FUNCTION_BLOCK DualHysteresis_AR_AX (* 2-way conversion of Analog to Digital with Hysteresis (Switch-on = MI +/- (ABS(DEAD) + ABS(HYSTERESIS)), Switch-off = MI +/- ABS(DEAD)) *)
  (* Standard: 61499-2; Description: Copyright (c) 2023 HR Agrartechnik GmbH This program and the accompanying materials are made available under the terms of the Eclipse Public License 2.0 which is available at https://www.eclipse.org/legal/epl-2.0/ SPDX-License-Identifier: EPL-2.0 *)
  (* Version 3.1, 2026-06-01, Gemini CLI, Addressed code review: absolute values for thresholds, explicit comparison semantics. *)
  (* Version 3.0, 2025-04-14, Patrick Aigner, changed package *)
  (* Version 1.0, 2023-06-06, Franz Höpfinger, HR Agrartechnik GmbH *)
  PACKAGE logiBUS::signalprocessing::hysteresis;
  IMPORT eclipse4diac::core::TypeHash;
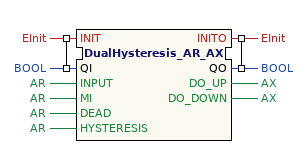
  EVENT_INPUT
    INIT : EInit WITH QI; (* Initialization Request *)
  END_EVENT
  EVENT_OUTPUT
    INITO : EInit WITH QO; (* Initialization Confirm *)
  END_EVENT
  VAR_INPUT
    QI : BOOL; (* Input event qualifier *)
  END_VAR
  VAR_OUTPUT
    QO : BOOL;
  END_VAR
  SOCKETS
    INPUT : adapter::types::unidirectional::AR; (* Input value *)
    MI : adapter::types::unidirectional::AR; (* Center point (e.g. 0.5 for 50%) *)
    DEAD : adapter::types::unidirectional::AR; (* Deadband around MI (absolute value). Switch-off points = MI +/- ABS(DEAD) *)
    HYSTERESIS : adapter::types::unidirectional::AR; (* Hysteresis value (absolute value). Switch-on points = MI +/- (ABS(DEAD) + ABS(HYSTERESIS)) *)
  END_SOCKETS
  PLUGS
    DO_UP : adapter::types::unidirectional::AX; (* UP *)
    DO_DOWN : adapter::types::unidirectional::AX; (* DOWN *)
  END_PLUGS
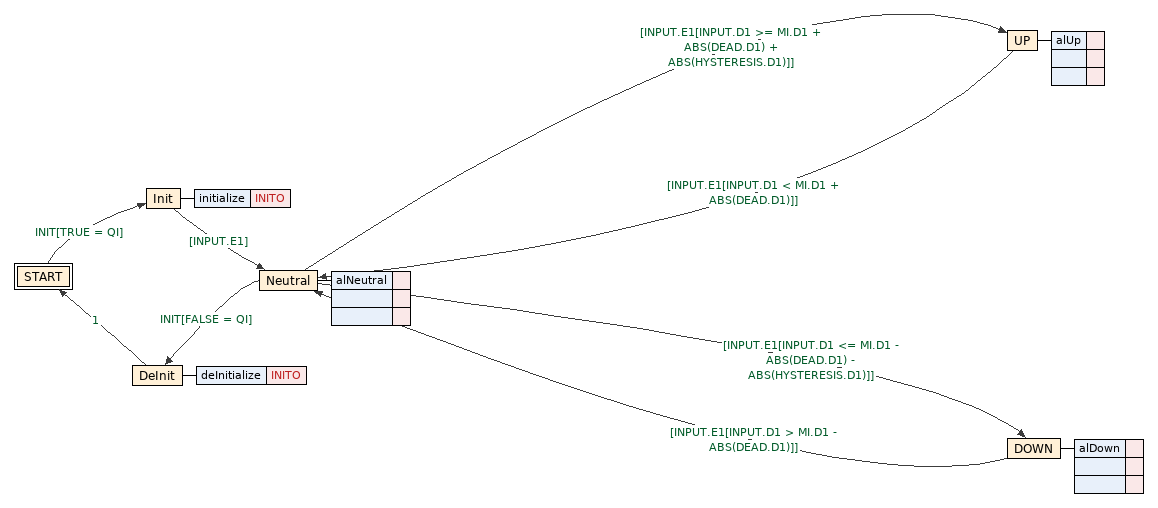
  EC_STATES
    START; (* Initial State *)
    Init : initialize -> INITO; (* Initialization *)
    UP : alUp; (* Normal execution *)
    Neutral : alNeutral;
    DeInit : deInitialize -> INITO;
    DOWN : alDown;
  END_STATES
  EC_TRANSITIONS
    START TO Init := INIT[TRUE = QI];
    Init TO Neutral := [INPUT.E1];
    Neutral TO DeInit := INIT[FALSE = QI];
    Neutral TO UP := [INPUT.E1[INPUT.D1 >= MI.D1 + ABS(DEAD.D1) + ABS(HYSTERESIS.D1)]]; (* Switch-on UP (inclusive) *)
    DeInit TO START := 1;
    Neutral TO DOWN := [INPUT.E1[INPUT.D1 <= MI.D1 - ABS(DEAD.D1) - ABS(HYSTERESIS.D1)]]; (* Switch-on DOWN (inclusive) *)
    DOWN TO Neutral := [INPUT.E1[INPUT.D1 > MI.D1 - ABS(DEAD.D1)]]; (* Switch-off DOWN (strict) *)
    UP TO Neutral := [INPUT.E1[INPUT.D1 < MI.D1 + ABS(DEAD.D1)]]; (* Switch-off UP (strict) *)
  END_TRANSITIONS
  ALGORITHM initialize IN ST:
QO := QI;
(* in any case go safe State *)
DO_UP.D1 := BOOL#FALSE;
DO_DOWN.D1 := BOOL#FALSE;
  END_ALGORITHM
  ALGORITHM deInitialize IN ST:
QO := BOOL#FALSE;
(* in any case go safe State *)
DO_UP.D1 := BOOL#FALSE;
DO_DOWN.D1 := BOOL#FALSE;
  END_ALGORITHM
  ALGORITHM alNeutral IN ST:
QO := QI;
(* in any case go safe State *)
DO_UP.D1 := BOOL#FALSE;
DO_DOWN.D1 := BOOL#FALSE;
  END_ALGORITHM
  ALGORITHM alUp IN ST:
QO := QI;
IF TRUE = QI THEN
	(* only perform normal operation of QI is true *)
	DO_UP.D1 := BOOL#TRUE;
	DO_DOWN.D1 := BOOL#FALSE;
END_IF;
  END_ALGORITHM
  ALGORITHM alDown IN ST:
QO := QI;
IF TRUE = QI THEN
	(* only perform normal operation of QI is true *)
	DO_UP.D1 := BOOL#FALSE;
	DO_DOWN.D1 := BOOL#TRUE;
END_IF;
  END_ALGORITHM
END_FUNCTION_BLOCK
